TYPE IoStatus :
STRUCT
	SensorStatus: SensorStatus;
	InputStatus: InputStatus;
END_STRUCT
END_TYPE

(* stored: Version 1.1.0.1, ProductVersion 3.1.4024.6
   DUT IoStatus: Id {7be4d157-f5c1-4063-a13d-ac0c63fd93f0} *)
